Universal Robots URScript: urcap_ros.script

def unnamed():
  set_safety_mode_transition_hardness(1)
  set_tool_voltage(0)
  step_count_f8b4a7b5_6e24_42e8_88a2_cde172f965e9 = 0.0
  thread Step_Counter_Thread_a18da4be_b2a1_4be3_be9c_1788a0db4eb5():
    while (True):
      step_count_f8b4a7b5_6e24_42e8_88a2_cde172f965e9 = step_count_f8b4a7b5_6e24_42e8_88a2_cde172f965e9 + 1.0
      sync()
    end
  end
  run Step_Counter_Thread_a18da4be_b2a1_4be3_be9c_1788a0db4eb5()
  set_tcp(p[0.0,0.0,0.0,0.0,0.0,0.0])
  set_payload(0.0)
  set_gravity([0.0, 0.0, 9.82])
  set_standard_analog_input_domain(0, 1)
  set_standard_analog_input_domain(1, 1)
  set_tool_analog_input_domain(0, 1)
  set_tool_analog_input_domain(1, 1)
  set_analog_outputdomain(0, 0)
  set_analog_outputdomain(1, 0)
  set_input_actions_to_default()
  # begin: URCap Installation Node
  #   Source: External Control, 1.0.5, FZI Research Center for Information Technology
  #   Type: External Control
  # end: URCap Installation Node
  while (True):
    $ 1 "Robot Program"
    # begin: URCap Program Node
    #   Source: External Control, 1.0.5, FZI Research Center for Information Technology
    #   Type: External Control
    $ 2 "Control by 192.168.56.1"
popup("The connection to the remote PC at 192.168.56.1:50002 could not be established. Reason: Connection refused (Connection refused)","Receive program failed", False, True, blocking=True)
sync()    # end: URCap Program Node
  end
end
